{attribute 'linkalways'} 
{attribute 'no_explicit_call' := 'This FB is a CLASS and must be accessed using methods or properties'}
{attribute 'enable_dynamic_creation'}
FUNCTION_BLOCK Node_F_VN_FindContours EXTENDS VisionNode
VAR
    ipSrcImage : _ITcVnImage;
    ipContours : _ITcVnContainer;
    hrPrev : _HRESULT(S_OK);
	hresult : _HRESULT(S_OK);
END_VAR

METHOD PUBLIC  Clone : I_Node
VAR
	pNode : POINTER TO Node_F_VN_FindContours;
END_VAR
pNode := __NEW(Node_F_VN_FindContours);
Clone := pNode^;
END_METHOD

METHOD FB_init : BOOL
VAR_INPUT
	bInitRetains : BOOL; // if TRUE, the retain variables are initialized (warm start / cold start)
	bInCopyCode : BOOL;  // if TRUE, the instance afterwards gets moved into the copy code (online change)
END_VAR
AddInput('ipSrcImage', ipSrcImage);
AddInput('hrPrev', hrPrev);
AddOutput('ipContours', ipContours);
AddOutput('hresult', hresult);
END_METHOD

METHOD PROTECTED OnExecute
hresult.Value := F_VN_FindContours(
	ipSrcImage := ipSrcImage.Value,
    ipContours := ipContours.Value,
	hrPrev:= hrPrev.Value);
END_METHOD

METHOD PUBLIC PreExecutionCheck
VAR_INPUT
	Check : I_PreExecutionChecks;
END_VAR
Check.IsTrue(ipSrcImage.IsValid, 'ipSrcImage must contain an image');
Check.IsTrue(ipSrcImage.HasChannelCount(1), 'ipSrcImage must contain 1 channel');
END_METHOD

END_FUNCTION_BLOCK

(* stored: Version 1.1.0.1, ProductVersion 3.1.4026.18
   POU Node_F_VN_FindContours: Id {7b30a029-3bbd-4901-86c1-2b5bb894aec5}, SpecialFunc None
   Folder Constructor: Id {3c3972cc-b449-4091-ae76-f8fab5823587}
   Method Clone: Id {0a233b80-2e16-43d7-ab26-c84bd961673a}
   Method FB_init: Id {954a0bc0-4a1c-49c7-b795-e82165143738}
   Method OnExecute: Id {4a41b4bd-1f7d-4cd3-86d0-5ffd9bba25ec}
   Method PreExecutionCheck: Id {b966ec77-caaf-4811-9a14-d5b3de74ffb1} *)
